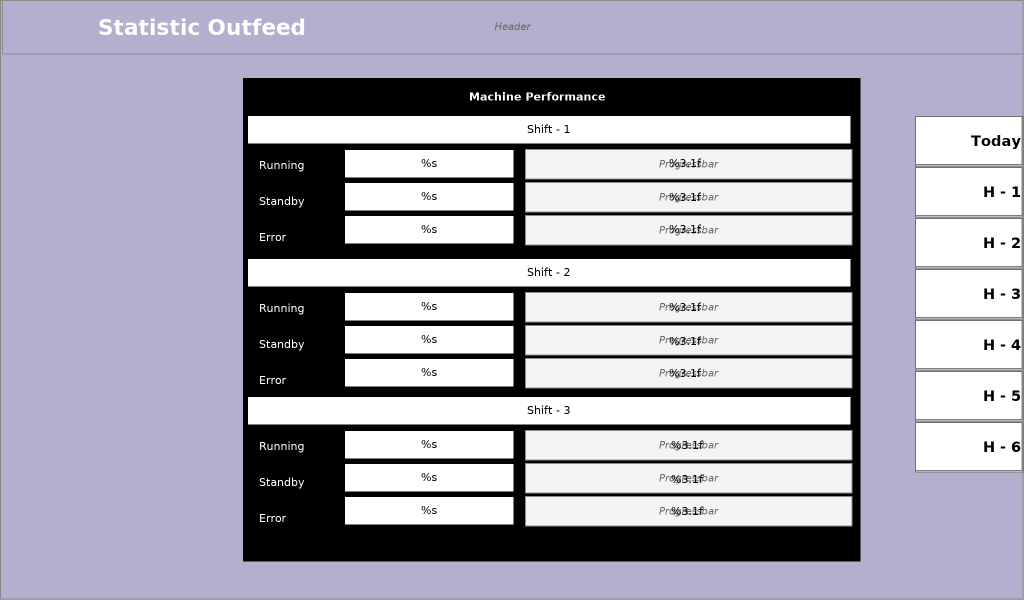
VISUALIZATION OEE_Outfeed  // 1024x600
    Frame (2,-1 1021x55)
        shows Header()
    RoundedRectangle (243,78 617x483)
    RoundedRectangle (247,115 604x29), "Shift - 1"
    Label (270,77 535x40), "Machine Performance"
    Label (256,148 78x35), "Running"
    Label (256,184 78x35), "Standby"
    Label (256,220 78x35), "Error"
    Progressbar (525,149 327x30), variable: Data_GVL.dt_OEEOutfeed.Precentage[0].Running
    Progressbar (525,182 327x30), variable: Data_GVL.dt_OEEOutfeed.Precentage[0].Stopped
    Progressbar (525,215 327x30), variable: Data_GVL.dt_OEEOutfeed.Precentage[0].Error
    RoundedRectangle (344,149 170x29), "%s", text variable: Data_GVL.dt_OEEOutfeed.HMI_Time[0].sRunning
    RoundedRectangle (344,182 170x29), "%s", text variable: Data_GVL.dt_OEEOutfeed.HMI_Time[0].sStopped
    RoundedRectangle (344,215 170x29), "%s", text variable: Data_GVL.dt_OEEOutfeed.HMI_Time[0].sError
    RoundedRectangle (247,258 604x29), "Shift - 2"
    Label (256,291 78x35), "Running"
    Label (256,327 78x35), "Standby"
    Label (256,363 78x35), "Error"
    Progressbar (525,292 327x30), variable: Data_GVL.dt_OEEOutfeed.Precentage[1].Running
    Progressbar (525,325 327x30), variable: Data_GVL.dt_OEEOutfeed.Precentage[1].Stopped
    Progressbar (525,358 327x30), variable: Data_GVL.dt_OEEOutfeed.Precentage[1].Error
    RoundedRectangle (344,292 170x29), "%s", text variable: Data_GVL.dt_OEEOutfeed.HMI_Time[1].sRunning
    RoundedRectangle (344,325 170x29), "%s", text variable: Data_GVL.dt_OEEOutfeed.HMI_Time[1].sStopped
    RoundedRectangle (344,358 170x29), "%s", text variable: Data_GVL.dt_OEEOutfeed.HMI_Time[1].sError
    RoundedRectangle (247,396 604x29), "Shift - 3"
    Label (256,429 78x35), "Running"
    Label (256,465 78x35), "Standby"
    Label (256,501 78x35), "Error"
    Progressbar (525,430 327x30), variable: Data_GVL.dt_OEEOutfeed.Precentage[2].Running
    Progressbar (525,463 327x30), variable: Data_GVL.dt_OEEOutfeed.Precentage[2].Stopped
    Progressbar (525,496 327x30), variable: Data_GVL.dt_OEEOutfeed.Precentage[2].Error
    RoundedRectangle (344,430 170x29), "%s", text variable: Data_GVL.dt_OEEOutfeed.HMI_Time[2].sRunning
    RoundedRectangle (344,463 170x29), "%s", text variable: Data_GVL.dt_OEEOutfeed.HMI_Time[2].sStopped
    RoundedRectangle (344,496 170x29), "%s", text variable: Data_GVL.dt_OEEOutfeed.HMI_Time[2].sError
    Button (915,116 109x50), "Today", image: VisuSymbols.Symbols.CalenderDay
        OnMouseClick: execute { Data_GVL.dt_OEEOutfeed.HMI_NumberPrev := 0; }
    Button (915,167 109x50), "H - 1", image: VisuSymbols.Symbols.CalenderDay
        OnMouseClick: execute { Data_GVL.dt_OEEOutfeed.HMI_NumberPrev := 1; }
    Button (915,218 109x50), "H - 2", image: VisuSymbols.Symbols.CalenderDay
        OnMouseClick: execute { Data_GVL.dt_OEEOutfeed.HMI_NumberPrev := 2; }
    Button (915,269 109x50), "H - 3", image: VisuSymbols.Symbols.CalenderDay
        OnMouseClick: execute { Data_GVL.dt_OEEOutfeed.HMI_NumberPrev := 3; }
    Button (915,320 109x50), "H - 4", image: VisuSymbols.Symbols.CalenderDay
        OnMouseClick: execute { Data_GVL.dt_OEEOutfeed.HMI_NumberPrev := 4; }
    Button (915,371 109x50), "H - 5", image: VisuSymbols.Symbols.CalenderDay
        OnMouseClick: execute { Data_GVL.dt_OEEOutfeed.HMI_NumberPrev := 5; }
    Button (915,422 109x50), "H - 6", image: VisuSymbols.Symbols.CalenderDay
        OnMouseClick: execute { Data_GVL.dt_OEEOutfeed.HMI_NumberPrev := 6; }
    RoundedRectangle (600,149 170x29), "%3.1f", text variable: Data_GVL.dt_OEEOutfeed.Precentage[0].Running
    RoundedRectangle (600,183 170x29), "%3.1f", text variable: Data_GVL.dt_OEEOutfeed.Precentage[0].Stopped
    RoundedRectangle (600,215 170x29), "%3.1f", text variable: Data_GVL.dt_OEEOutfeed.Precentage[0].Error
    RoundedRectangle (600,293 170x29), "%3.1f", text variable: Data_GVL.dt_OEEOutfeed.Precentage[1].Running
    RoundedRectangle (600,327 170x29), "%3.1f", text variable: Data_GVL.dt_OEEOutfeed.Precentage[1].Stopped
    RoundedRectangle (600,359 170x29), "%3.1f", text variable: Data_GVL.dt_OEEOutfeed.Precentage[1].Error
    RoundedRectangle (602,431 170x29), "%3.1f", text variable: Data_GVL.dt_OEEOutfeed.Precentage[2].Running
    RoundedRectangle (602,465 170x29), "%3.1f", text variable: Data_GVL.dt_OEEOutfeed.Precentage[2].Stopped
    RoundedRectangle (602,497 170x29), "%3.1f", text variable: Data_GVL.dt_OEEOutfeed.Precentage[2].Error
    Label (95,15 214x25), "Statistic Outfeed"
END_VISUALIZATION

(* stored: Version 1.1.0.1, ProductVersion 3.1.4024.12
   Visu OEE_Outfeed: Id {2001434d-7949-4720-95ee-0b58db8b7699} *)
